Fanuc KAREL source: ko00034.KL

PROGRAM KO00034
%STACKSIZE=65535
%PRIORITY=65535
%NOLOCKGROUP
VAR
P1 : POSITION
P2 : POSITION
F : BOOLEAN
OUT : XYZWPR
BEGIN
F=TRUE
-- UNSAFE_SOURCE_IR line 11: OUT = MIRROR(convert_position_to_xyzwprext(P1), P2, F)
END KO00034
